FUNCTION_BLOCK CALC_ABSOLUTE_VALUE
VAR_INPUT
    IN_VAL : INT;
END_VAR

VAR_OUTPUT
    OUT_VAL : INT;
    STATUS  : INT;   (* 0 indicates successful operation; 1 indicates that saturation occurred due to an overflow risk *)
END_VAR

(* Calculate the absolute value using INT arithmetic.
   If IN_VAL equals the lowest representable INT value, its negation would exceed the permitted range.
   In that case, we saturate the output to the maximum INT value (32767) and set an error status. *)
IF IN_VAL = (-32767 - 1) THEN
    OUT_VAL := 32767;
    STATUS  := 1;
ELSIF IN_VAL < 0 THEN
    OUT_VAL := -IN_VAL;
    STATUS  := 0;
ELSE
    OUT_VAL := IN_VAL;
    STATUS  := 0;
END_IF;

END_FUNCTION_BLOCK